(* CODESYS project GVL_TEST_IO.gvl.xml

Project tree, tasks and I/O mapping:
  global variables GVL_TEST_IO
*)

// GVL_TEST_IO
{attribute 'qualified_only'}
VAR_GLOBAL
	// Логический вход. Физический адрес назначается отдельно в Device I/O Mapping CODESYS.
	xSc500BenchKeyInput : BOOL := FALSE;
END_VAR
